KUKA KRL program: Work_2.src, Work_2.dat

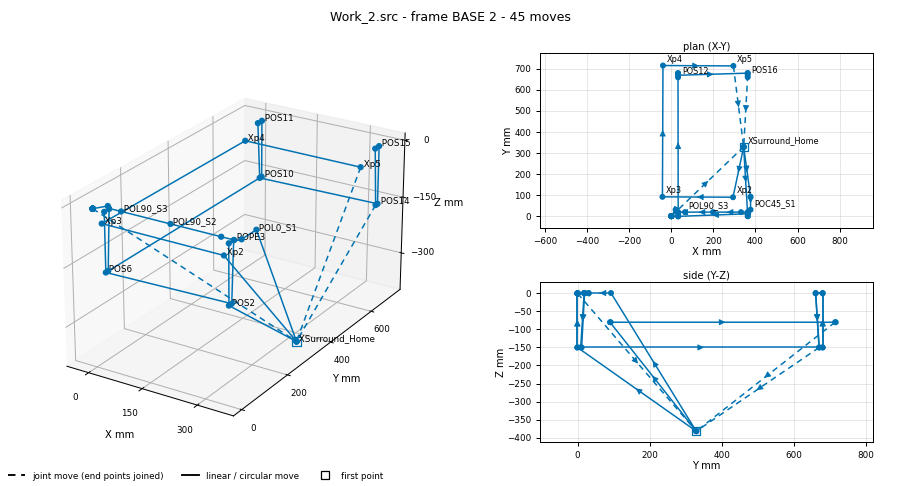
[picture p0: tool path of Work_2.src in frame BASE 2, 45 of 45 moves have a stored position in this frame; points joined in program order, loops and branches not executed]
--- Work_2.src ---
&ACCESS RVP
&REL 333
&PARAM EDITMASK = *
&PARAM TEMPLATE = C:\KRC\Roboter\Template\vorgabe
&PARAM DISKPATH = KRC:\R1\Program\HG
DEF Work_2( )
;FOLD INI;%{PE}
  ;FOLD BASISTECH INI
    GLOBAL INTERRUPT DECL 3 WHEN $STOPMESS==TRUE DO IR_STOPM ( )
    INTERRUPT ON 3
    BAS (#INITMOV,0 )
  ;ENDFOLD (BASISTECH INI)
  ;FOLD USER INI
    ;Make your modifications here

  ;ENDFOLD (USER INI)
;ENDFOLD (INI)

;FOLD Vision.Vision_Ini ;%{PE}%MKUKATPUSER




EKRL_Vision_Int_Data("Xml_Ini_Data")


;ENDFOLD
;loop
;FOLD PTP Surround_Home Vel=20 % PDAT1 Tool[2]:Work_Tool Base[2]:B_2;%{PE}%R 8.3.48,%MKUKATPBASIS,%CMOVE,%VPTP,%P 1:PTP, 2:Surround_Home, 3:, 5:20, 7:PDAT1
$BWDSTART=FALSE
PDAT_ACT=PPDAT1
FDAT_ACT=FSurround_Home
BAS(#PTP_PARAMS,20)
PTP XSurround_Home
;ENDFOLD

;FOLD Vision.Camera_Offset Camera_NAME :P2, Area:45, Work:2;%{PE}%MKUKATPUSER

 HanGao_Camera_Offset(#Calibration ,1,2,XP2)





;ENDFOLD
;FOLD LIN p2 Vel=.3 m/s CPDAT1 Tool[2]:Work_Tool Base[2]:B_2;%{PE}%R 8.3.48,%MKUKATPBASIS,%CMOVE,%VLIN,%P 1:LIN, 2:p2, 3:, 5:.3, 7:CPDAT1
$BWDSTART=FALSE
LDAT_ACT=LCPDAT1
FDAT_ACT=Fp2
BAS(#CP_PARAMS,.3)
LIN Xp2
;ENDFOLD
;FOLD Vision.Find_Model Work:2, Area:45;%{PE}%MKUKATPUSER



EKRL_Find_Model_Send("Xml_Vision_Model",2,1)



;ENDFOLD


;FOLD Vision.Camera_Offset Camera_NAME :P3, Area:135, Work:2;%{PE}%MKUKATPUSER

 HanGao_Camera_Offset(#Calibration ,2,2,XP3)





;ENDFOLD
;FOLD LIN p3 Vel=.3 m/s CPDAT2 Tool[2]:Work_Tool Base[2]:B_2;%{PE}%R 8.3.48,%MKUKATPBASIS,%CMOVE,%VLIN,%P 1:LIN, 2:p3, 3:, 5:.3, 7:CPDAT2
$BWDSTART=FALSE
LDAT_ACT=LCPDAT2
FDAT_ACT=Fp3
BAS(#CP_PARAMS,.3)
LIN Xp3
;ENDFOLD
;FOLD Vision.Find_Model Work:2, Area:135;%{PE}%MKUKATPUSER



EKRL_Find_Model_Send("Xml_Vision_Model",2,2)



;ENDFOLD


;FOLD Vision.Camera_Offset Camera_NAME :P4, Area:225, Work:2;%{PE}%MKUKATPUSER

 HanGao_Camera_Offset(#Calibration ,3,2,XP4)





;ENDFOLD
;FOLD LIN p4 Vel=.3 m/s CPDAT3 Tool[2]:Work_Tool Base[2]:B_2;%{PE}%R 8.3.48,%MKUKATPBASIS,%CMOVE,%VLIN,%P 1:LIN, 2:p4, 3:, 5:.3, 7:CPDAT3
$BWDSTART=FALSE
LDAT_ACT=LCPDAT3
FDAT_ACT=Fp4
BAS(#CP_PARAMS,.3)
LIN Xp4
;ENDFOLD
;FOLD Vision.Find_Model Work:2, Area:225;%{PE}%MKUKATPUSER



EKRL_Find_Model_Send("Xml_Vision_Model",2,3)



;ENDFOLD


;FOLD Vision.Camera_Offset Camera_NAME :P5, Area:315, Work:2;%{PE}%MKUKATPUSER

 HanGao_Camera_Offset(#Calibration ,4,2,XP5)





;ENDFOLD
;FOLD LIN p5 Vel=.3 m/s CPDAT4 Tool[2]:Work_Tool Base[2]:B_2;%{PE}%R 8.3.48,%MKUKATPBASIS,%CMOVE,%VLIN,%P 1:LIN, 2:p5, 3:, 5:.3, 7:CPDAT4
$BWDSTART=FALSE
LDAT_ACT=LCPDAT4
FDAT_ACT=Fp5
BAS(#CP_PARAMS,.3)
LIN Xp5
;ENDFOLD
;FOLD Vision.Find_Model Work:2, Area:315;%{PE}%MKUKATPUSER



EKRL_Find_Model_Send("Xml_Vision_Model",2,4)



;ENDFOLD
;endloop
;halt
;FOLD PTP Surround_Home Vel=10 % PDAT4 Tool[2]:Work_Tool Base[2]:B_2;%{PE}%R 8.3.48,%MKUKATPBASIS,%CMOVE,%VPTP,%P 1:PTP, 2:Surround_Home, 3:, 5:10, 7:PDAT4
$BWDSTART=FALSE
PDAT_ACT=PPDAT4
FDAT_ACT=FSurround_Home
BAS(#PTP_PARAMS,10)
PTP XSurround_Home
;ENDFOLD
;FOLD Surround_LIN.S_LIN Point:L0_S1, Vel=.2m/s, Point: 90/%, Area:LO, LDAT:L0_L1, OFFSET_NO:1, Work: N_2;%{PE}%MKUKATPUSER

; LIN L0_S1POS: X=0, Y=0, Z=0, A=0, B=0, C=0
; LIN Offset POS:X=0, Y=0, Z=0
HanGao_Surr_Calculate( 90, #L0, #L_LIN_POS , POL0_S1, , , L0_Welding_Craft[2,1].Welding_Offset  , , 1, 2 )

LL0_L1.VEL=L0_Welding_Craft[2,1].Welding_Speed
LL0_L1.ACC=L0_Welding_Craft[2,1].Welding_ACC
LL0_L1.APO_DIST=L0_Welding_Craft[2,1].Welding_CDIS

FDAT_ACT=FL0_S1
LDAT_ACT=LL0_L1
BAS(#CP_PARAMS,L0_Welding_Craft[2,1].Welding_Speed )
LIN POL0_S1 C_DIS C_DIS

;ENDFOLD
;FOLD Laser_Function.LSON POW= .9%, Sec= 0S;%{PE}%MKUKATPUSER


  $ANOUT[1]= .9
  LSON(0)


;ENDFOLD
;FOLD Surround_LIN.S_C_LIN Point:C45_S1, Vel=.04m/s, Area: C45, LDAT:C45_L1, Work: N_2;%{PE}%MKUKATPUSER

; CIR C45_S1POS: X=0, Y=0, Z=0, A=0, B=0, C=0
; CIR Offset POS:X=0, Y=0, Z=0
HanGao_Surr_Calculate(  , #C45, #C_LIN_POS , POC45_S1, , , C45_Welding_Craft[2,1].Welding_Offset , ,  , 2)

LC45_L1.VEL=C45_Welding_Craft[2,1].Welding_Speed
LC45_L1.ACC=C45_Welding_Craft[2,1].Welding_ACC
LC45_L1.APO_DIST=C45_Welding_Craft[2,1].Welding_CDIS

FDAT_ACT=FC45_S1
LDAT_ACT=LC45_L1
BAS(#CP_PARAMS, C45_Welding_Craft[2,1].Welding_Speed )
LIN POC45_S1 C_DIS C_DIS

;ENDFOLD
;FOLD Surround_CIR.S_C_CIR Point:PM3, PE3, Vel=.04m/s, Angle Area: C45, Work: N_2;%{PE}%MKUKATPUSER

; CIR MID POS:PM3 : X=0, Y=0, Z=0, A=0, B=0, C=0
; CIR END POS:PE3 : X=0, Y=0, Z=0, A=0, B=0, C=0
; CIR_MID_OFFSET  : X=0, Y=0, Z=0
; CIR_END_OFFSET  : X=0, Y=.3, Z=0
HanGao_Surr_Calculate(  , #C45, #C_CIR_POS ,  , POPM3, POPE3 , C45_Welding_Craft[2,2].Welding_Offset  , C45_Welding_Craft[2, 3].Welding_Offset  ,  , 2)

LPM3.VEL=C45_Welding_Craft[2,3].Welding_Speed
LPM3.ACC=C45_Welding_Craft[2,3].Welding_ACC
LPM3.APO_DIST=C45_Welding_Craft[2,3].Welding_CDIS

FDAT_ACT=FPE3
LDAT_ACT=LPM3
BAS(#CP_PARAMS,C45_Welding_Craft[2,3].Welding_Speed )
CIRC POPM3, POPE3 C_DIS C_DIS

;ENDFOLD
;FOLD Surround_LIN.S_LIN Point:L90_S1, Vel=.04m/s, Point: 10/%, Area:L90, LDAT:L90_L1, OFFSET_NO:1, Work: N_2;%{PE}%MKUKATPUSER

; LIN L90_S1POS: X=0, Y=0, Z=0, A=0, B=0, C=0
; LIN Offset POS:X=0, Y=.2, Z=0
HanGao_Surr_Calculate( 10, #L90, #L_LIN_POS , POL90_S1, , , L90_Welding_Craft[2,1].Welding_Offset  , , 1, 2 )

LL90_L1.VEL=L90_Welding_Craft[2,1].Welding_Speed
LL90_L1.ACC=L90_Welding_Craft[2,1].Welding_ACC
LL90_L1.APO_DIST=L90_Welding_Craft[2,1].Welding_CDIS

FDAT_ACT=FL90_S1
LDAT_ACT=LL90_L1
BAS(#CP_PARAMS,L90_Welding_Craft[2,1].Welding_Speed )
LIN POL90_S1 C_DIS C_DIS

;ENDFOLD
;FOLD Surround_LIN.S_LIN Point:L90_S2, Vel=.04m/s, Point: 50/%, Area:L90, LDAT:L90_L2, OFFSET_NO:2, Work: N_2;%{PE}%MKUKATPUSER

; LIN L90_S2POS: X=198.086502, Y=19.0685, Z=1, A=0, B=0, C=20
; LIN Offset POS:X=0, Y=.2, Z=0
HanGao_Surr_Calculate( 50, #L90, #L_LIN_POS , POL90_S2, , , L90_Welding_Craft[2,2].Welding_Offset  , , 2, 2 )

LL90_L2.VEL=L90_Welding_Craft[2,2].Welding_Speed
LL90_L2.ACC=L90_Welding_Craft[2,2].Welding_ACC
LL90_L2.APO_DIST=L90_Welding_Craft[2,2].Welding_CDIS

FDAT_ACT=FL90_S2
LDAT_ACT=LL90_L2
BAS(#CP_PARAMS,L90_Welding_Craft[2,2].Welding_Speed )
LIN POL90_S2 C_DIS C_DIS

;ENDFOLD
;FOLD Surround_LIN.S_LIN Point:L90_S3, Vel=.04m/s, Point: 90/%, Area:L90, LDAT:L90_L3, OFFSET_NO:3, Work: N_2;%{PE}%MKUKATPUSER

; LIN L90_S3POS: X=64.8645, Y=19.0867844, Z=1, A=0, B=0, C=20
; LIN Offset POS:X=0, Y=.2, Z=0
HanGao_Surr_Calculate( 90, #L90, #L_LIN_POS , POL90_S3, , , L90_Welding_Craft[2,3].Welding_Offset  , , 3, 2 )

LL90_L3.VEL=L90_Welding_Craft[2,3].Welding_Speed
LL90_L3.ACC=L90_Welding_Craft[2,3].Welding_ACC
LL90_L3.APO_DIST=L90_Welding_Craft[2,3].Welding_CDIS

FDAT_ACT=FL90_S3
LDAT_ACT=LL90_L3
BAS(#CP_PARAMS,L90_Welding_Craft[2,3].Welding_Speed )
LIN POL90_S3 C_DIS C_DIS

;ENDFOLD
;FOLD Surround_LIN.S_C_LIN Point:C135_S1, Vel=.04m/s, Area: C135, LDAT:C135_L1, Work: N_2;%{PE}%MKUKATPUSER

; CIR C135_S1POS: X=31.5589905, Y=18.8913536, Z=1, A=0, B=0, C=20
; CIR Offset POS:X=0, Y=.2, Z=0
HanGao_Surr_Calculate(  , #C135, #C_LIN_POS , POC135_S1, , , C135_Welding_Craft[2,1].Welding_Offset , ,  , 2)

LC135_L1.VEL=C135_Welding_Craft[2,1].Welding_Speed
LC135_L1.ACC=C135_Welding_Craft[2,1].Welding_ACC
LC135_L1.APO_DIST=C135_Welding_Craft[2,1].Welding_CDIS

FDAT_ACT=FC135_S1
LDAT_ACT=LC135_L1
BAS(#CP_PARAMS, C135_Welding_Craft[2,1].Welding_Speed )
LIN POC135_S1 C_DIS C_DIS

;ENDFOLD
;FOLD Surround_CIR.S_C_CIR Point:PM4, PE4, Vel=.04m/s, Angle Area: C135, Work: N_2;%{PE}%MKUKATPUSER

; CIR MID POS:PM4 : X=22.393, Y=22.49, Z=1, A=0, B=0, C=0
; CIR END POS:PE4 : X=20.0512314, Y=30.8929977, Z=0, A=0, B=-20, C=0
; CIR_MID_OFFSET  : X=0, Y=0, Z=0
; CIR_END_OFFSET  : X=.5, Y=0, Z=-1
HanGao_Surr_Calculate(  , #C135, #C_CIR_POS ,  , POPM4, POPE4 , C135_Welding_Craft[2,2].Welding_Offset  , C135_Welding_Craft[2, 3].Welding_Offset  ,  , 2)

LPM4.VEL=C135_Welding_Craft[2,3].Welding_Speed
LPM4.ACC=C135_Welding_Craft[2,3].Welding_ACC
LPM4.APO_DIST=C135_Welding_Craft[2,3].Welding_CDIS

FDAT_ACT=FPE4
LDAT_ACT=LPM4
BAS(#CP_PARAMS,C135_Welding_Craft[2,3].Welding_Speed )
CIRC POPM4, POPE4 C_DIS C_DIS

;ENDFOLD
;FOLD Surround_LIN.S_LIN Point:L180_S1, Vel=.04m/s, Point: 10/%, Area:L180, LDAT:L180_L1, OFFSET_NO:1, Work: N_2;%{PE}%MKUKATPUSER

; LIN L180_S1POS: X=19.5112858, Y=92.5949936, Z=0, A=0, B=-20, C=0
; LIN Offset POS:X=0, Y=0, Z=-1
HanGao_Surr_Calculate( 10, #L180, #L_LIN_POS , POL180_S1, , , L180_Welding_Craft[2,1].Welding_Offset  , , 1, 2 )

LL180_L1.VEL=L180_Welding_Craft[2,1].Welding_Speed
LL180_L1.ACC=L180_Welding_Craft[2,1].Welding_ACC
LL180_L1.APO_DIST=L180_Welding_Craft[2,1].Welding_CDIS

FDAT_ACT=FL180_S1
LDAT_ACT=LL180_L1
BAS(#CP_PARAMS,L180_Welding_Craft[2,1].Welding_Speed )
LIN POL180_S1 C_DIS C_DIS

;ENDFOLD
;FOLD Surround_LIN.S_LIN Point:L180_S2, Vel=.04m/s, Point: 50/%, Area:L180, LDAT:L180_L2, OFFSET_NO:2, Work: N_2;%{PE}%MKUKATPUSER

; LIN L180_S2POS: X=0, Y=0, Z=0, A=0, B=0, C=0
; LIN Offset POS:X=0, Y=0, Z=-1
HanGao_Surr_Calculate( 50, #L180, #L_LIN_POS , POL180_S2, , , L180_Welding_Craft[2,2].Welding_Offset  , , 2, 2 )

LL180_L2.VEL=L180_Welding_Craft[2,2].Welding_Speed
LL180_L2.ACC=L180_Welding_Craft[2,2].Welding_ACC
LL180_L2.APO_DIST=L180_Welding_Craft[2,2].Welding_CDIS

FDAT_ACT=FL180_S2
LDAT_ACT=LL180_L2
BAS(#CP_PARAMS,L180_Welding_Craft[2,2].Welding_Speed )
LIN POL180_S2 C_DIS C_DIS

;ENDFOLD
;FOLD Surround_LIN.S_LIN Point:L180_S3, Vel=.04m/s, Point: 95/%, Area:L180, LDAT:L180_L3, OFFSET_NO:3, Work: N_2;%{PE}%MKUKATPUSER

; LIN L180_S3POS: X=0, Y=0, Z=0, A=0, B=0, C=0
; LIN Offset POS:X=.5, Y=0, Z=-1
HanGao_Surr_Calculate( 95, #L180, #L_LIN_POS , POL180_S3, , , L180_Welding_Craft[2,3].Welding_Offset  , , 3, 2 )

LL180_L3.VEL=L180_Welding_Craft[2,3].Welding_Speed
LL180_L3.ACC=L180_Welding_Craft[2,3].Welding_ACC
LL180_L3.APO_DIST=L180_Welding_Craft[2,3].Welding_CDIS

FDAT_ACT=FL180_S3
LDAT_ACT=LL180_L3
BAS(#CP_PARAMS,L180_Welding_Craft[2,3].Welding_Speed )
LIN POL180_S3 C_DIS C_DIS

;ENDFOLD
;FOLD Surround_LIN.S_C_LIN Point:C225_S1, Vel=.04m/s, Area: C225, LDAT:C225_L1, Work: N_2;%{PE}%MKUKATPUSER

; CIR C225_S1POS: X=0, Y=0, Z=0, A=0, B=0, C=0
; CIR Offset POS:X=.5, Y=0, Z=-1
HanGao_Surr_Calculate(  , #C225, #C_LIN_POS , POC225_S1, , , C225_Welding_Craft[2,1].Welding_Offset , ,  , 2)

LC225_L1.VEL=C225_Welding_Craft[2,1].Welding_Speed
LC225_L1.ACC=C225_Welding_Craft[2,1].Welding_ACC
LC225_L1.APO_DIST=C225_Welding_Craft[2,1].Welding_CDIS

FDAT_ACT=FC225_S1
LDAT_ACT=LC225_L1
BAS(#CP_PARAMS, C225_Welding_Craft[2,1].Welding_Speed )
LIN POC225_S1 C_DIS C_DIS

;ENDFOLD
;FOLD Surround_CIR.S_C_CIR Point:PM5, PE5, Vel=.04m/s, Angle Area: C225, Work: N_2;%{PE}%MKUKATPUSER

; CIR MID POS:PM5 : X=22.393, Y=22.49, Z=1, A=0, B=0, C=0
; CIR END POS:PE5 : X=20.0512314, Y=30.8929977, Z=0, A=0, B=-20, C=0
; CIR_MID_OFFSET  : X=0, Y=0, Z=0
; CIR_END_OFFSET  : X=.5, Y=0, Z=-1
HanGao_Surr_Calculate(  , #C225, #C_CIR_POS ,  , POPM5, POPE5 , C225_Welding_Craft[2,2].Welding_Offset  , C225_Welding_Craft[2, 3].Welding_Offset  ,  , 2)

LPM5.VEL=C225_Welding_Craft[2,3].Welding_Speed
LPM5.ACC=C225_Welding_Craft[2,3].Welding_ACC
LPM5.APO_DIST=C225_Welding_Craft[2,3].Welding_CDIS

FDAT_ACT=FPE5
LDAT_ACT=LPM5
BAS(#CP_PARAMS,C225_Welding_Craft[2,3].Welding_Speed )
CIRC POPM5, POPE5 C_DIS C_DIS

;ENDFOLD
;FOLD Surround_LIN.S_LIN Point:L270_S1, Vel=.04m/s, Point: 10/%, Area:L270, LDAT:l270_L1, OFFSET_NO:1, Work: N_2;%{PE}%MKUKATPUSER

; LIN L270_S1POS: X=0, Y=0, Z=0, A=0, B=0, C=0
; LIN Offset POS:X=0, Y=0, Z=-1
HanGao_Surr_Calculate( 10, #L270, #L_LIN_POS , POL270_S1, , , L270_Welding_Craft[2,1].Welding_Offset  , , 1, 2 )

Ll270_L1.VEL=L270_Welding_Craft[2,1].Welding_Speed
Ll270_L1.ACC=L270_Welding_Craft[2,1].Welding_ACC
Ll270_L1.APO_DIST=L270_Welding_Craft[2,1].Welding_CDIS

FDAT_ACT=FL270_S1
LDAT_ACT=Ll270_L1
BAS(#CP_PARAMS,L270_Welding_Craft[2,1].Welding_Speed )
LIN POL270_S1 C_DIS C_DIS

;ENDFOLD
;FOLD Surround_LIN.S_LIN Point:L270_S2, Vel=.04m/s, Point: 50/%, Area:L270, LDAT:L270_L2, OFFSET_NO:2, Work: N_2;%{PE}%MKUKATPUSER

; LIN L270_S2POS: X=0, Y=0, Z=0, A=0, B=0, C=0
; LIN Offset POS:X=0, Y=0, Z=0
HanGao_Surr_Calculate( 50, #L270, #L_LIN_POS , POL270_S2, , , L270_Welding_Craft[2,2].Welding_Offset  , , 2, 2 )

LL270_L2.VEL=L270_Welding_Craft[2,2].Welding_Speed
LL270_L2.ACC=L270_Welding_Craft[2,2].Welding_ACC
LL270_L2.APO_DIST=L270_Welding_Craft[2,2].Welding_CDIS

FDAT_ACT=FL270_S2
LDAT_ACT=LL270_L2
BAS(#CP_PARAMS,L270_Welding_Craft[2,2].Welding_Speed )
LIN POL270_S2 C_DIS C_DIS

;ENDFOLD
;FOLD Surround_LIN.S_LIN Point:L270_S3, Vel=.04m/s, Point: 95/%, Area:L270, LDAT:L270_L3, OFFSET_NO:3, Work: N_2;%{PE}%MKUKATPUSER

; LIN L270_S3POS: X=0, Y=0, Z=0, A=0, B=0, C=0
; LIN Offset POS:X=0, Y=-.8, Z=0
HanGao_Surr_Calculate( 95, #L270, #L_LIN_POS , POL270_S3, , , L270_Welding_Craft[2,3].Welding_Offset  , , 3, 2 )

LL270_L3.VEL=L270_Welding_Craft[2,3].Welding_Speed
LL270_L3.ACC=L270_Welding_Craft[2,3].Welding_ACC
LL270_L3.APO_DIST=L270_Welding_Craft[2,3].Welding_CDIS

FDAT_ACT=FL270_S3
LDAT_ACT=LL270_L3
BAS(#CP_PARAMS,L270_Welding_Craft[2,3].Welding_Speed )
LIN POL270_S3 C_DIS C_DIS

;ENDFOLD
;FOLD Surround_LIN.S_C_LIN Point:C315_S1, Vel=.04m/s, Area: C315, LDAT:C315_L1, Work: N_2;%{PE}%MKUKATPUSER

; CIR C315_S1POS: X=0, Y=0, Z=0, A=0, B=0, C=0
; CIR Offset POS:X=0, Y=-.8, Z=0
HanGao_Surr_Calculate(  , #C315, #C_LIN_POS , POC315_S1, , , C315_Welding_Craft[2,1].Welding_Offset , ,  , 2)

LC315_L1.VEL=C315_Welding_Craft[2,1].Welding_Speed
LC315_L1.ACC=C315_Welding_Craft[2,1].Welding_ACC
LC315_L1.APO_DIST=C315_Welding_Craft[2,1].Welding_CDIS

FDAT_ACT=FC315_S1
LDAT_ACT=LC315_L1
BAS(#CP_PARAMS, C315_Welding_Craft[2,1].Welding_Speed )
LIN POC315_S1 C_DIS C_DIS

;ENDFOLD
;FOLD Surround_CIR.S_C_CIR Point:PM7, PE7, Vel=.04m/s, Angle Area: C315, Work: N_2;%{PE}%MKUKATPUSER

; CIR MID POS:PM7 : X=0, Y=0, Z=0, A=0, B=0, C=0
; CIR END POS:PE7 : X=0, Y=0, Z=0, A=0, B=0, C=0
; CIR_MID_OFFSET  : X=0, Y=0, Z=0
; CIR_END_OFFSET  : X=0, Y=.5, Z=0
HanGao_Surr_Calculate(  , #C315, #C_CIR_POS ,  , POPM7, POPE7 , C315_Welding_Craft[2,2].Welding_Offset  , C315_Welding_Craft[2, 3].Welding_Offset  ,  , 2)

LPM7.VEL=C315_Welding_Craft[2,3].Welding_Speed
LPM7.ACC=C315_Welding_Craft[2,3].Welding_ACC
LPM7.APO_DIST=C315_Welding_Craft[2,3].Welding_CDIS

FDAT_ACT=FPE7
LDAT_ACT=LPM7
BAS(#CP_PARAMS,C315_Welding_Craft[2,3].Welding_Speed )
CIRC POPM7, POPE7 C_DIS C_DIS

;ENDFOLD
;FOLD Surround_LIN.S_LIN Point:L0_S2, Vel=.04m/s, Point: 10/%, Area:LO, LDAT:L0_L2, OFFSET_NO:2, Work: N_2;%{PE}%MKUKATPUSER

; LIN L0_S2POS: X=0, Y=0, Z=0, A=0, B=0, C=0
; LIN Offset POS:X=0, Y=0, Z=0
HanGao_Surr_Calculate( 10, #L0, #L_LIN_POS , POL0_S2, , , L0_Welding_Craft[2,2].Welding_Offset  , , 2, 2 )

LL0_L2.VEL=L0_Welding_Craft[2,2].Welding_Speed
LL0_L2.ACC=L0_Welding_Craft[2,2].Welding_ACC
LL0_L2.APO_DIST=L0_Welding_Craft[2,2].Welding_CDIS

FDAT_ACT=FL0_S2
LDAT_ACT=LL0_L2
BAS(#CP_PARAMS,L0_Welding_Craft[2,2].Welding_Speed )
LIN POL0_S2 C_DIS C_DIS

;ENDFOLD
;FOLD Surround_LIN.S_LIN Point:L0_S3, Vel=.04m/s, Point: 50/%, Area:LO, LDAT:L0_L3, OFFSET_NO:3, Work: N_2;%{PE}%MKUKATPUSER

; LIN L0_S3POS: X=0, Y=0, Z=0, A=0, B=0, C=0
; LIN Offset POS:X=0, Y=0, Z=0
HanGao_Surr_Calculate( 50, #L0, #L_LIN_POS , POL0_S3, , , L0_Welding_Craft[2,3].Welding_Offset  , , 3, 2 )

LL0_L3.VEL=L0_Welding_Craft[2,3].Welding_Speed
LL0_L3.ACC=L0_Welding_Craft[2,3].Welding_ACC
LL0_L3.APO_DIST=L0_Welding_Craft[2,3].Welding_CDIS

FDAT_ACT=FL0_S3
LDAT_ACT=LL0_L3
BAS(#CP_PARAMS,L0_Welding_Craft[2,3].Welding_Speed )
LIN POL0_S3 C_DIS C_DIS

;ENDFOLD
;FOLD Surround_LIN.S_LIN Point:L0_S4, Vel=.04m/s, Point: 95/%, Area:LO, LDAT:L0_L4, OFFSET_NO:4, Work: N_2;%{PE}%MKUKATPUSER

; LIN L0_S4POS: X=0, Y=0, Z=0, A=0, B=0, C=0
; LIN Offset POS:X=0, Y=0, Z=0
HanGao_Surr_Calculate( 95, #L0, #L_LIN_POS , POL0_S4, , , L0_Welding_Craft[2,4].Welding_Offset  , , 4, 2 )

LL0_L4.VEL=L0_Welding_Craft[2,4].Welding_Speed
LL0_L4.ACC=L0_Welding_Craft[2,4].Welding_ACC
LL0_L4.APO_DIST=L0_Welding_Craft[2,4].Welding_CDIS

FDAT_ACT=FL0_S4
LDAT_ACT=LL0_L4
BAS(#CP_PARAMS,L0_Welding_Craft[2,4].Welding_Speed )
LIN POL0_S4 C_DIS C_DIS

;ENDFOLD
LSOFF()


;FOLD PTP Surround_Home Vel=10 % PDAT2 Tool[2]:Work_Tool Base[2]:B_2;%{PE}%R 8.3.48,%MKUKATPBASIS,%CMOVE,%VPTP,%P 1:PTP, 2:Surround_Home, 3:, 5:10, 7:PDAT2
$BWDSTART=FALSE
PDAT_ACT=PPDAT2
FDAT_ACT=FSurround_Home
BAS(#PTP_PARAMS,10)
PTP XSurround_Home
;ENDFOLD
if (false) THEN
;halt
;return
;FOLD Short_Craft.S_LIN Point:S2, Vel=.1m/s, Area: N45, Short_Pos: Safety, Point: 50/%, LDAT:L2, Work: N_2;%{PE}%MKUKATPUSER

; LIN S2POS: X=364.543579, Y=6.21706629, Z=0, A=0, B=0, C=0
; LIN Offset POS:X=0, Y=0, Z=0
HanGao_Surr_Calculate( 50, #N45, #L_LIN_POS , POS2, , , N45_Short_Craft[2,1].Welding_Offset  , , 1, 2, N2_Sink_Data.Sink_Type)

FDAT_ACT=FS2
LDAT_ACT=LL2
BAS(#CP_PARAMS,N45_Short_Craft[2,1].Welding_Speed )
LIN POS2 C_DIS C_DIS

;ENDFOLD
;FOLD Short_Craft.S_LIN Point:S3, Vel=.1m/s, Area: N45, Short_Pos: Start, Point: 50/%, LDAT:L3, Work: N_2;%{PE}%MKUKATPUSER

; LIN S3POS: X=0, Y=0, Z=0, A=0, B=0, C=0
; LIN Offset POS:X=0, Y=0, Z=0
HanGao_Surr_Calculate( 50, #N45, #L_LIN_POS , POS3, , , N45_Short_Craft[2,2].Welding_Offset  , , 2, 2, N2_Sink_Data.Sink_Type)

FDAT_ACT=FS3
LDAT_ACT=LL3
BAS(#CP_PARAMS,N45_Short_Craft[2,2].Welding_Speed )
LIN POS3 C_DIS C_DIS

;ENDFOLD
;FOLD ANOUT AO01=.6 ;%{PE}%R 8.3.48,%MKUKATPBASIS,%CANA,%VANOUT_STAT,%P 2:CHANNEL_1, 4:.6
$ANOUT[1]=.6
;ENDFOLD
LSON()
;FOLD Short_Craft.S_LIN Point:S4, Vel=.1m/s, Area: N45, Short_Pos: End, Point: 50/%, LDAT:L4, Work: N_2;%{PE}%MKUKATPUSER

; LIN S4POS: X=364.543579, Y=6.21706629, Z=0, A=0, B=0, C=0
; LIN Offset POS:X=0, Y=0, Z=0
HanGao_Surr_Calculate( 50, #N45, #L_LIN_POS , POS4, , , N45_Short_Craft[2,3].Welding_Offset  , , 3, 2, N2_Sink_Data.Sink_Type)

FDAT_ACT=FS4
LDAT_ACT=LL4
BAS(#CP_PARAMS,N45_Short_Craft[2,3].Welding_Speed )
LIN POS4 C_DIS C_DIS

;ENDFOLD
;FOLD Short_Craft.S_LIN Point:S5, Vel=.1m/s, Area: N45, Short_Pos: BackWelding, Point: 10/%, LDAT:L5, Work: N_2;%{PE}%MKUKATPUSER

; LIN S5POS: X=364.551483, Y=29.6448097, Z=0, A=0, B=0, C=0
; LIN Offset POS:X=0, Y=0, Z=0
HanGao_Surr_Calculate( 10, #N45, #L_LIN_POS , POS5, , , N45_Short_Craft[2,4].Welding_Offset  , , 4, 2, N2_Sink_Data.Sink_Type)

FDAT_ACT=FS5
LDAT_ACT=LL5
BAS(#CP_PARAMS,N45_Short_Craft[2,4].Welding_Speed )
LIN POS5 C_DIS C_DIS

;ENDFOLD
LSOFF()


;FOLD Short_Craft.S_LIN Point:S6, Vel=.1m/s, Area: N135, Short_Pos: Safety, Point: 50/%, LDAT:L6, Work: N_2;%{PE}%MKUKATPUSER

; LIN S6POS: X=364.547089, Y=16.5598412, Z=-150, A=0, B=0, C=0
; LIN Offset POS:X=0, Y=0, Z=0
HanGao_Surr_Calculate( 50, #N135, #L_LIN_POS , POS6, , , N135_Short_Craft[2,1].Welding_Offset  , , 1, 2, N2_Sink_Data.Sink_Type)

FDAT_ACT=FS6
LDAT_ACT=LL6
BAS(#CP_PARAMS,N135_Short_Craft[2,1].Welding_Speed )
LIN POS6 C_DIS C_DIS

;ENDFOLD
;FOLD Short_Craft.S_LIN Point:S7, Vel=.1m/s, Area: N135, Short_Pos: Start, Point: 50/%, LDAT:L7, Work: N_2;%{PE}%MKUKATPUSER

; LIN S7POS: X=36.6399193, Y=6.3348074, Z=-150, A=0, B=0, C=0
; LIN Offset POS:X=0, Y=0, Z=0
HanGao_Surr_Calculate( 50, #N135, #L_LIN_POS , POS7, , , N135_Short_Craft[2,2].Welding_Offset  , , 2, 2, N2_Sink_Data.Sink_Type)

FDAT_ACT=FS7
LDAT_ACT=LL7
BAS(#CP_PARAMS,N135_Short_Craft[2,2].Welding_Speed )
LIN POS7 C_DIS C_DIS

;ENDFOLD
;FOLD ANOUT AO01=.6 ;%{PE}%R 8.3.48,%MKUKATPBASIS,%CANA,%VANOUT_STAT,%P 2:CHANNEL_1, 4:.6
$ANOUT[1]=.6
;ENDFOLD
LSON()
;FOLD Short_Craft.S_LIN Point:S8, Vel=.1m/s, Area: N135, Short_Pos: End, Point: 50/%, LDAT:L8, Work: N_2;%{PE}%MKUKATPUSER

; LIN S8POS: X=36.6399193, Y=6.3348074, Z=0, A=0, B=0, C=0
; LIN Offset POS:X=0, Y=0, Z=0
HanGao_Surr_Calculate( 50, #N135, #L_LIN_POS , POS8, , , N135_Short_Craft[2,3].Welding_Offset  , , 3, 2, N2_Sink_Data.Sink_Type)

FDAT_ACT=FS8
LDAT_ACT=LL8
BAS(#CP_PARAMS,N135_Short_Craft[2,3].Welding_Speed )
LIN POS8 C_DIS C_DIS

;ENDFOLD
;FOLD Short_Craft.S_LIN Point:S9, Vel=.1m/s, Area: N135, Short_Pos: BackWelding, Point: 50/%, LDAT:L9, Work: N_2;%{PE}%MKUKATPUSER

; LIN S9POS: X=36.5802116, Y=29.963192, Z=0, A=0, B=0, C=0
; LIN Offset POS:X=0, Y=0, Z=0
HanGao_Surr_Calculate( 50, #N135, #L_LIN_POS , POS9, , , N135_Short_Craft[2,4].Welding_Offset  , , 4, 2, N2_Sink_Data.Sink_Type)

FDAT_ACT=FS9
LDAT_ACT=LL9
BAS(#CP_PARAMS,N135_Short_Craft[2,4].Welding_Speed )
LIN POS9 C_DIS C_DIS

;ENDFOLD
LSOFF()


;FOLD Short_Craft.S_LIN Point:S10, Vel=.1m/s, Area: N225, Short_Pos: Safety, Point: 50/%, LDAT:L10, Work: N_2;%{PE}%MKUKATPUSER

; LIN S10POS: X=36.6100655, Y=18.1489983, Z=-150, A=0, B=0, C=0
; LIN Offset POS:X=0, Y=0, Z=0
HanGao_Surr_Calculate( 50, #N225, #L_LIN_POS , POS10, , , N225_Short_Craft[2,1].Welding_Offset  , , 1, 2, N2_Sink_Data.Sink_Type)

FDAT_ACT=FS10
LDAT_ACT=LL10
BAS(#CP_PARAMS,N225_Short_Craft[2,1].Welding_Speed )
LIN POS10 C_DIS C_DIS

;ENDFOLD
;FOLD Short_Craft.S_LIN Point:S11, Vel=.1m/s, Area: N225, Short_Pos: Start, Point: 50/%, LDAT:L11, Work: N_2;%{PE}%MKUKATPUSER

; LIN S11POS: X=46.8049, Y=687.557678, Z=-150, A=0, B=0, C=0
; LIN Offset POS:X=0, Y=0, Z=0
HanGao_Surr_Calculate( 50, #N225, #L_LIN_POS , POS11, , , N225_Short_Craft[2,2].Welding_Offset  , , 2, 2, N2_Sink_Data.Sink_Type)

FDAT_ACT=FS11
LDAT_ACT=LL11
BAS(#CP_PARAMS,N225_Short_Craft[2,2].Welding_Speed )
LIN POS11 C_DIS C_DIS

;ENDFOLD
;FOLD ANOUT AO01=.6 ;%{PE}%R 8.3.48,%MKUKATPBASIS,%CANA,%VANOUT_STAT,%P 2:CHANNEL_1, 4:.6
$ANOUT[1]=.6
;ENDFOLD
LSON()
;FOLD Short_Craft.S_LIN Point:S12, Vel=.1m/s, Area: N225, Short_Pos: End, Point: 50/%, LDAT:L12, Work: N_2;%{PE}%MKUKATPUSER

; LIN S12POS: X=46.8049, Y=687.557678, Z=0, A=0, B=0, C=0
; LIN Offset POS:X=0, Y=0, Z=0
HanGao_Surr_Calculate( 50, #N225, #L_LIN_POS , POS12, , , N225_Short_Craft[2,3].Welding_Offset  , , 3, 2, N2_Sink_Data.Sink_Type)

FDAT_ACT=FS12
LDAT_ACT=LL12
BAS(#CP_PARAMS,N225_Short_Craft[2,3].Welding_Speed )
LIN POS12 C_DIS C_DIS

;ENDFOLD
;FOLD Short_Craft.S_LIN Point:S13, Vel=.1m/s, Area: N225, Short_Pos: BackWelding, Point: 50/%, LDAT:L13, Work: N_2;%{PE}%MKUKATPUSER

; LIN S13POS: X=46.2807388, Y=663.904114, Z=0, A=0, B=0, C=0
; LIN Offset POS:X=0, Y=0, Z=0
HanGao_Surr_Calculate( 50, #N225, #L_LIN_POS , POS13, , , N225_Short_Craft[2,4].Welding_Offset  , , 4, 2, N2_Sink_Data.Sink_Type)

FDAT_ACT=FS13
LDAT_ACT=LL13
BAS(#CP_PARAMS,N225_Short_Craft[2,4].Welding_Speed )
LIN POS13 C_DIS C_DIS

;ENDFOLD
LSOFF()


;FOLD Short_Craft.S_LIN Point:S14, Vel=.1m/s, Area: N315, Short_Pos: Safety, Point: 50/%, LDAT:L14, Work: N_2;%{PE}%MKUKATPUSER

; LIN S14POS: X=46.54282, Y=675.730896, Z=-150, A=0, B=0, C=0
; LIN Offset POS:X=0, Y=0, Z=0
HanGao_Surr_Calculate( 50, #N315, #L_LIN_POS , POS14, , , N315_Short_Craft[2,1].Welding_Offset  , , 1, 2, N2_Sink_Data.Sink_Type)

FDAT_ACT=FS14
LDAT_ACT=LL14
BAS(#CP_PARAMS,N315_Short_Craft[2,1].Welding_Speed )
LIN POS14 C_DIS C_DIS

;ENDFOLD
;FOLD Short_Craft.S_LIN Point:S15, Vel=.1m/s, Area: N315, Short_Pos: Start, Point: 50/%, LDAT:L15, Work: N_2;%{PE}%MKUKATPUSER

; LIN S15POS: X=375.074402, Y=680.748169, Z=-150, A=0, B=0, C=0
; LIN Offset POS:X=0, Y=0, Z=0
HanGao_Surr_Calculate( 50, #N315, #L_LIN_POS , POS15, , , N315_Short_Craft[2,2].Welding_Offset  , , 2, 2, N2_Sink_Data.Sink_Type)

FDAT_ACT=FS15
LDAT_ACT=LL15
BAS(#CP_PARAMS,N315_Short_Craft[2,2].Welding_Speed )
LIN POS15 C_DIS C_DIS

;ENDFOLD
;FOLD ANOUT AO01=.6 ;%{PE}%R 8.3.48,%MKUKATPBASIS,%CANA,%VANOUT_STAT,%P 2:CHANNEL_1, 4:.6
$ANOUT[1]=.6
;ENDFOLD
LSON()
;FOLD Short_Craft.S_LIN Point:S16, Vel=.1m/s, Area: N315, Short_Pos: End, Point: 50/%, LDAT:L16, Work: N_2;%{PE}%MKUKATPUSER

; LIN S16POS: X=375.074402, Y=680.748169, Z=0, A=0, B=0, C=0
; LIN Offset POS:X=0, Y=0, Z=0
HanGao_Surr_Calculate( 50, #N315, #L_LIN_POS , POS16, , , N315_Short_Craft[2,3].Welding_Offset  , , 3, 2, N2_Sink_Data.Sink_Type)

FDAT_ACT=FS16
LDAT_ACT=LL16
BAS(#CP_PARAMS,N315_Short_Craft[2,3].Welding_Speed )
LIN POS16 C_DIS C_DIS

;ENDFOLD
;FOLD Short_Craft.S_LIN Point:S17, Vel=.1m/s, Area: N315, Short_Pos: BackWelding, Point: 50/%, LDAT:L17, Work: N_2;%{PE}%MKUKATPUSER

; LIN S17POS: X=374.424377, Y=657.20105, Z=0, A=0, B=0, C=0
; LIN Offset POS:X=0, Y=0, Z=0
HanGao_Surr_Calculate( 50, #N315, #L_LIN_POS , POS17, , , N315_Short_Craft[2,4].Welding_Offset  , , 4, 2, N2_Sink_Data.Sink_Type)

FDAT_ACT=FS17
LDAT_ACT=LL17
BAS(#CP_PARAMS,N315_Short_Craft[2,4].Welding_Speed )
LIN POS17 C_DIS C_DIS

;ENDFOLD
LSOFF()
endif

;FOLD PTP Surround_Home CONT Vel=30 % PDAT3 Tool[2]:Work_Tool Base[2]:B_2;%{PE}%R 8.3.48,%MKUKATPBASIS,%CMOVE,%VPTP,%P 1:PTP, 2:Surround_Home, 3:C_DIS, 5:30, 7:PDAT3
$BWDSTART=FALSE
PDAT_ACT=PPDAT3
FDAT_ACT=FSurround_Home
BAS(#PTP_PARAMS,30)
PTP XSurround_Home C_DIS
;ENDFOLD
END

--- Work_2.dat ---
&ACCESS RVP
&REL 333
&PARAM EDITMASK = *
&PARAM TEMPLATE = C:\KRC\Roboter\Template\vorgabe
&PARAM DISKPATH = KRC:\R1\Program\HG
DEFDAT  Work_2
;FOLD EXTERNAL DECLARATIONS;%{PE}%MKUKATPBASIS,%CEXT,%VCOMMON,%P
;FOLD BASISTECH EXT;%{PE}%MKUKATPBASIS,%CEXT,%VEXT,%P
EXT  BAS (BAS_COMMAND  :IN,REAL  :IN )
DECL INT SUCCESS
;ENDFOLD (BASISTECH EXT)
;FOLD USER EXT;%{E}%MKUKATPUSER,%CEXT,%VEXT,%P
;Make your modifications here

;ENDFOLD (USER EXT)
;ENDFOLD (EXTERNAL DECLARATIONS)
DECL BASIS_SUGG_T LAST_BASIS={POINT1[] "P0                      ",POINT2[] "P0                      ",CP_PARAMS[] "CPDAT0                  ",PTP_PARAMS[] "PDAT0                   ",CONT[] "                        ",CP_VEL[] "2.0                     ",PTP_VEL[] " 100                    ",SYNC_PARAMS[] "SYNCDAT                 ",SPL_NAME[] "S0                      ",A_PARAMS[] "ADAT0                   "}
DECL E6POS XSURROUND_HOME={X 343.780548,Y 329.155823,Z -382.275,A 0.441927075,B -0.0416149125,C -0.0704164580,S 2,T 10,E1 0.0,E2 0.0,E3 0.0,E4 0.0,E5 0.0,E6 0.0}
DECL FDAT FSurround_Home={TOOL_NO 2,BASE_NO 2,IPO_FRAME #BASE,POINT2[] " ",TQ_STATE FALSE}
DECL PDAT PPDAT1={VEL 100.000,ACC 20.0000,APO_DIST 100.000,GEAR_JERK 50.0000,EXAX_IGN 0}
DECL PDAT PPDAT2={VEL 100.000,ACC 20.0000,APO_DIST 100.000,GEAR_JERK 50.0000,EXAX_IGN 0}
DECL E6POS POS2={X 363.220,Y -0.316000,Z -150.000,A 0.0,B 0.0,C 0.0}
DECL FDAT FS2={TOOL_NO 2,BASE_NO 2,IPO_FRAME #BASE,POINT2[] " ",TQ_STATE FALSE}
DECL LDAT LL2={VEL 0.100000,ACC 100.000,APO_DIST 5.00000,APO_FAC 50.0000,AXIS_VEL 100.000,AXIS_ACC 100.000,ORI_TYP #VAR,CIRC_TYP #BASE,JERK_FAC 50.0000,GEAR_JERK 50.0000,EXAX_IGN 0}
DECL E6POS POS3={X 363.220,Y -0.316000,Z 0.0,A 0.0,B 0.0,C 0.0}
DECL FDAT FS3={TOOL_NO 2,BASE_NO 2,IPO_FRAME #BASE,POINT2[] " ",TQ_STATE FALSE}
DECL LDAT LL3={VEL 0.100000,ACC 100.000,APO_DIST 0.0,APO_FAC 50.0000,AXIS_VEL 100.000,AXIS_ACC 100.000,ORI_TYP #VAR,CIRC_TYP #BASE,JERK_FAC 50.0000,GEAR_JERK 50.0000,EXAX_IGN 0}
DECL E6POS POS4={X 363.395,Y 19.3140,Z 0.0,A 0.0,B 0.0,C 0.0}
DECL FDAT FS4={TOOL_NO 2,BASE_NO 2,IPO_FRAME #BASE,POINT2[] " ",TQ_STATE FALSE}
DECL LDAT LL4={VEL 0.100000,ACC 100.000,APO_DIST 0.0,APO_FAC 50.0000,AXIS_VEL 100.000,AXIS_ACC 100.000,ORI_TYP #VAR,CIRC_TYP #BASE,JERK_FAC 50.0000,GEAR_JERK 50.0000,EXAX_IGN 0}
DECL E6POS POS5={X 363.323059,Y 11.2466183,Z -150.000,A 0.0,B 0.0,C 0.0}
DECL FDAT FS5={TOOL_NO 2,BASE_NO 2,IPO_FRAME #BASE,POINT2[] " ",TQ_STATE FALSE}
DECL LDAT LL5={VEL 0.100000,ACC 100.000,APO_DIST 0.0,APO_FAC 50.0000,AXIS_VEL 100.000,AXIS_ACC 100.000,ORI_TYP #VAR,CIRC_TYP #BASE,JERK_FAC 50.0000,GEAR_JERK 50.0000,EXAX_IGN 0}
DECL E6POS POPM3={X 373.063,Y 22.4860,Z 1.00000,A 0.0,B 0.0,C 0.0}
DECL E6POS POPE3={X 364.614,Y 19.1456451,Z 1.00000,A 0.0,B 0.0,C 20.0000}
DECL FDAT FPE3={TOOL_NO 2,BASE_NO 2,IPO_FRAME #BASE,POINT2[] " ",TQ_STATE FALSE}
DECL LDAT LPM3={VEL 0.01000000,ACC 100.000,APO_DIST 5.00000,APO_FAC 50.0000,AXIS_VEL 100.000,AXIS_ACC 100.000,ORI_TYP #VAR,CIRC_TYP #BASE,JERK_FAC 50.0000,GEAR_JERK 50.0000,EXAX_IGN 0}
DECL E6POS POS6={X 32.5260,Y -0.971000,Z -150.000,A 0.0,B 0.0,C 0.0}
DECL FDAT FS6={TOOL_NO 2,BASE_NO 2,IPO_FRAME #BASE,POINT2[] " ",TQ_STATE FALSE}
DECL LDAT LL6={VEL 0.100000,ACC 100.000,APO_DIST 0.0,APO_FAC 50.0000,AXIS_VEL 100.000,AXIS_ACC 100.000,ORI_TYP #VAR,CIRC_TYP #BASE,JERK_FAC 50.0000,GEAR_JERK 50.0000,EXAX_IGN 0}
DECL E6POS POS7={X 32.5260,Y -0.971000,Z 0.0,A 0.0,B 0.0,C 0.0}
DECL FDAT FS7={TOOL_NO 2,BASE_NO 2,IPO_FRAME #BASE,POINT2[] " ",TQ_STATE FALSE}
DECL LDAT LL7={VEL 0.100000,ACC 100.000,APO_DIST 0.0,APO_FAC 50.0000,AXIS_VEL 100.000,AXIS_ACC 100.000,ORI_TYP #VAR,CIRC_TYP #BASE,JERK_FAC 50.0000,GEAR_JERK 50.0000,EXAX_IGN 0}
DECL E6POS POS8={X 32.3940,Y 18.1940,Z 0.0,A 0.0,B 0.0,C 0.0}
DECL FDAT FS8={TOOL_NO 2,BASE_NO 2,IPO_FRAME #BASE,POINT2[] " ",TQ_STATE FALSE}
DECL LDAT LL8={VEL 0.100000,ACC 100.000,APO_DIST 0.0,APO_FAC 50.0000,AXIS_VEL 100.000,AXIS_ACC 100.000,ORI_TYP #VAR,CIRC_TYP #BASE,JERK_FAC 50.0000,GEAR_JERK 50.0000,EXAX_IGN 0}
DECL E6POS POS9={X 32.4600,Y 8.61150074,Z -150.000,A 0.0,B 0.0,C 0.0}
DECL FDAT FS9={TOOL_NO 2,BASE_NO 2,IPO_FRAME #BASE,POINT2[] " ",TQ_STATE FALSE}
DECL LDAT LL9={VEL 0.100000,ACC 100.000,APO_DIST 0.0,APO_FAC 50.0000,AXIS_VEL 100.000,AXIS_ACC 100.000,ORI_TYP #VAR,CIRC_TYP #BASE,JERK_FAC 50.0000,GEAR_JERK 50.0000,EXAX_IGN 0}
DECL E6POS POPM4={X 22.3930,Y 22.4900,Z 1.00000,A 0.0,B 0.0,C 0.0}
DECL E6POS POPE4={X 20.0512314,Y 30.8929977,Z 0.0,A 0.0,B -20.0000,C 0.0}
DECL FDAT FPE4={TOOL_NO 2,BASE_NO 2,IPO_FRAME #BASE,POINT2[] " ",TQ_STATE FALSE}
DECL LDAT LPM4={VEL 0.0120000,ACC 100.000,APO_DIST 5.00000,APO_FAC 50.0000,AXIS_VEL 100.000,AXIS_ACC 100.000,ORI_TYP #VAR,CIRC_TYP #BASE,JERK_FAC 50.0000,GEAR_JERK 50.0000,EXAX_IGN 0}
DECL E6POS POPM5={X 0.0,Y 0.0,Z 0.0,A 0.0,B 0.0,C 0.0}
DECL E6POS POPE5={X 0.0,Y 0.0,Z 0.0,A 0.0,B 0.0,C 0.0}
DECL FDAT FPE5={TOOL_NO 2,BASE_NO 2,IPO_FRAME #BASE,POINT2[] " ",TQ_STATE FALSE}
DECL LDAT LPM5={VEL 0.0400000,ACC 100.000,APO_DIST 5.00000,APO_FAC 50.0000,AXIS_VEL 100.000,AXIS_ACC 100.000,ORI_TYP #VAR,CIRC_TYP #BASE,JERK_FAC 50.0000,GEAR_JERK 50.0000,EXAX_IGN 0}
DECL E6POS POPM7={X 0.0,Y 0.0,Z 0.0,A 0.0,B 0.0,C 0.0}
DECL E6POS POPE7={X 0.0,Y 0.0,Z 0.0,A 0.0,B 0.0,C 0.0}
DECL FDAT FPE7={TOOL_NO 2,BASE_NO 2,IPO_FRAME #BASE,POINT2[] " ",TQ_STATE FALSE}
DECL LDAT LPM7={VEL 0.0400000,ACC 100.000,APO_DIST 5.00000,APO_FAC 50.0000,AXIS_VEL 100.000,AXIS_ACC 100.000,ORI_TYP #VAR,CIRC_TYP #BASE,JERK_FAC 50.0000,GEAR_JERK 50.0000,EXAX_IGN 0}
DECL E6POS POS10={X 31.6330,Y 679.439,Z -150.000,A 0.0,B 0.0,C 0.0}
DECL FDAT FS10={TOOL_NO 2,BASE_NO 2,IPO_FRAME #BASE,POINT2[] " ",TQ_STATE FALSE}
DECL LDAT LL10={VEL 0.100000,ACC 100.000,APO_DIST 0.0,APO_FAC 50.0000,AXIS_VEL 100.000,AXIS_ACC 100.000,ORI_TYP #VAR,CIRC_TYP #BASE,JERK_FAC 50.0000,GEAR_JERK 50.0000,EXAX_IGN 0}
DECL E6POS POS11={X 31.6330,Y 679.439,Z 0.0,A 0.0,B 0.0,C 0.0}
DECL FDAT FS11={TOOL_NO 2,BASE_NO 2,IPO_FRAME #BASE,POINT2[] " ",TQ_STATE FALSE}
DECL LDAT LL11={VEL 0.100000,ACC 100.000,APO_DIST 0.0,APO_FAC 50.0000,AXIS_VEL 100.000,AXIS_ACC 100.000,ORI_TYP #VAR,CIRC_TYP #BASE,JERK_FAC 50.0000,GEAR_JERK 50.0000,EXAX_IGN 0}
DECL E6POS POS12={X 31.8670,Y 660.025,Z 0.0,A 0.0,B 0.0,C 0.0}
DECL FDAT FS12={TOOL_NO 2,BASE_NO 2,IPO_FRAME #BASE,POINT2[] " ",TQ_STATE FALSE}
DECL LDAT LL12={VEL 0.100000,ACC 100.000,APO_DIST 0.0,APO_FAC 50.0000,AXIS_VEL 100.000,AXIS_ACC 100.000,ORI_TYP #VAR,CIRC_TYP #BASE,JERK_FAC 50.0000,GEAR_JERK 50.0000,EXAX_IGN 0}
DECL E6POS POS13={X 31.7500,Y 669.732056,Z -150.000,A 0.0,B 0.0,C 0.0}
DECL FDAT FS13={TOOL_NO 2,BASE_NO 2,IPO_FRAME #BASE,POINT2[] " ",TQ_STATE FALSE}
DECL LDAT LL13={VEL 0.100000,ACC 100.000,APO_DIST 0.0,APO_FAC 50.0000,AXIS_VEL 100.000,AXIS_ACC 100.000,ORI_TYP #VAR,CIRC_TYP #BASE,JERK_FAC 50.0000,GEAR_JERK 50.0000,EXAX_IGN 0}
DECL E6POS POS14={X 362.986,Y 679.910,Z -150.000,A 0.0,B 0.0,C 0.0}
DECL FDAT FS14={TOOL_NO 2,BASE_NO 2,IPO_FRAME #BASE,POINT2[] " ",TQ_STATE FALSE}
DECL LDAT LL14={VEL 0.100000,ACC 100.000,APO_DIST 0.0,APO_FAC 50.0000,AXIS_VEL 100.000,AXIS_ACC 100.000,ORI_TYP #VAR,CIRC_TYP #BASE,JERK_FAC 50.0000,GEAR_JERK 50.0000,EXAX_IGN 0}
DECL E6POS POS15={X 362.986,Y 679.910,Z 1.00000,A 0.0,B 0.0,C 0.0}
DECL FDAT FS15={TOOL_NO 2,BASE_NO 2,IPO_FRAME #BASE,POINT2[] " ",TQ_STATE FALSE}
DECL LDAT LL15={VEL 0.100000,ACC 100.000,APO_DIST 0.0,APO_FAC 50.0000,AXIS_VEL 100.000,AXIS_ACC 100.000,ORI_TYP #VAR,CIRC_TYP #BASE,JERK_FAC 50.0000,GEAR_JERK 50.0000,EXAX_IGN 0}
DECL E6POS POS16={X 363.044,Y 660.468,Z 1.00000,A 0.0,B 0.0,C 0.0}
DECL FDAT FS16={TOOL_NO 2,BASE_NO 2,IPO_FRAME #BASE,POINT2[] " ",TQ_STATE FALSE}
DECL LDAT LL16={VEL 0.100000,ACC 100.000,APO_DIST 0.0,APO_FAC 50.0000,AXIS_VEL 100.000,AXIS_ACC 100.000,ORI_TYP #VAR,CIRC_TYP #BASE,JERK_FAC 50.0000,GEAR_JERK 50.0000,EXAX_IGN 0}
DECL E6POS POS17={X 363.015,Y 670.188965,Z -150.000,A 0.0,B 0.0,C 0.0}
DECL FDAT FS17={TOOL_NO 2,BASE_NO 2,IPO_FRAME #BASE,POINT2[] " ",TQ_STATE FALSE}
DECL LDAT LL17={VEL 0.100000,ACC 100.000,APO_DIST 0.0,APO_FAC 50.0000,AXIS_VEL 100.000,AXIS_ACC 100.000,ORI_TYP #VAR,CIRC_TYP #BASE,JERK_FAC 50.0000,GEAR_JERK 50.0000,EXAX_IGN 0}
DECL PDAT PPDAT3={VEL 100.000,ACC 20.0000,APO_DIST 100.000,APO_MODE #CDIS,GEAR_JERK 50.0000,EXAX_IGN 0}
DECL FDAT FL0_S2={TOOL_NO 2,BASE_NO 2,IPO_FRAME #BASE,POINT2[] " ",TQ_STATE FALSE}
DECL E6POS POL0_S2={X 0.0,Y 0.0,Z 0.0,A 0.0,B 0.0,C 0.0}
DECL FDAT FL0={TOOL_NO 2,BASE_NO 11,IPO_FRAME #BASE,POINT2[] " ",TQ_STATE FALSE}
DECL E6POS POL0_s4={X 0.0,Y 0.0,Z 0.0,A 0.0,B 0.0,C 0.0}
DECL FDAT FL0_s4={TOOL_NO 2,BASE_NO 2,IPO_FRAME #BASE,POINT2[] " ",TQ_STATE FALSE}
DECL E6POS POC45_S5={X 404.000,Y 36.0000,Z -1.00000,A 0.0,B 20.0000,C 0.0}
DECL FDAT FC45_S5={TOOL_NO 2,BASE_NO 11,IPO_FRAME #BASE,POINT2[] " ",TQ_STATE FALSE}
DECL E6POS POL0_S1={X 376.526398,Y 92.6378174,Z 1.00000,A 0.0,B 20.0000,C 0.0}
DECL FDAT FL0_S1={TOOL_NO 2,BASE_NO 2,IPO_FRAME #BASE,POINT2[] " ",TQ_STATE FALSE}
DECL E6POS POC45_S1={X 376.599762,Y 30.8439941,Z 1.00000,A 0.0,B 20.0000,C 0.0}
DECL FDAT FC45_S1={TOOL_NO 2,BASE_NO 2,IPO_FRAME #BASE,POINT2[] " ",TQ_STATE FALSE}
DECL LDAT LL0_L1={VEL 0.200000,ACC 50.0000,APO_DIST 5.00000,APO_FAC 50.0000,AXIS_VEL 100.000,AXIS_ACC 100.000,ORI_TYP #VAR,CIRC_TYP #BASE,JERK_FAC 50.0000,GEAR_JERK 50.0000,EXAX_IGN 0}
DECL LDAT LC45_L1={VEL 0.0250000,ACC 100.000,APO_DIST 5.00000,APO_FAC 50.0000,AXIS_VEL 100.000,AXIS_ACC 100.000,ORI_TYP #VAR,CIRC_TYP #BASE,JERK_FAC 50.0000,GEAR_JERK 50.0000,EXAX_IGN 0}
DECL E6POS POL90_S1={X 331.308502,Y 19.0502167,Z 1.00000,A 0.0,B 0.0,C 20.0000}
DECL FDAT FL90_S1={TOOL_NO 2,BASE_NO 2,IPO_FRAME #BASE,POINT2[] " ",TQ_STATE FALSE}
DECL LDAT LL90_L1={VEL 0.0250000,ACC 100.000,APO_DIST 5.00000,APO_FAC 50.0000,AXIS_VEL 100.000,AXIS_ACC 100.000,ORI_TYP #VAR,CIRC_TYP #BASE,JERK_FAC 50.0000,GEAR_JERK 50.0000,EXAX_IGN 0}
DECL E6POS POL90_S2={X 198.086502,Y 19.0685,Z 1.00000,A 0.0,B 0.0,C 20.0000}
DECL FDAT FL90_S2={TOOL_NO 2,BASE_NO 2,IPO_FRAME #BASE,POINT2[] " ",TQ_STATE FALSE}
DECL LDAT LL90_L2={VEL 0.0250000,ACC 100.000,APO_DIST 5.00000,APO_FAC 50.0000,AXIS_VEL 100.000,AXIS_ACC 100.000,ORI_TYP #VAR,CIRC_TYP #BASE,JERK_FAC 50.0000,GEAR_JERK 50.0000,EXAX_IGN 0}
DECL E6POS POL90_S3={X 64.8645,Y 19.0867844,Z 1.00000,A 0.0,B 0.0,C 20.0000}
DECL FDAT FL90_S3={TOOL_NO 2,BASE_NO 2,IPO_FRAME #BASE,POINT2[] " ",TQ_STATE FALSE}
DECL LDAT LL90_L3={VEL 0.0250000,ACC 100.000,APO_DIST 5.00000,APO_FAC 50.0000,AXIS_VEL 100.000,AXIS_ACC 100.000,ORI_TYP #VAR,CIRC_TYP #BASE,JERK_FAC 50.0000,GEAR_JERK 50.0000,EXAX_IGN 0}
DECL E6POS POC135_S1={X 31.5589905,Y 18.8913536,Z 1.00000,A 0.0,B 0.0,C 20.0000}
DECL FDAT FC135_S1={TOOL_NO 2,BASE_NO 2,IPO_FRAME #BASE,POINT2[] " ",TQ_STATE FALSE}
DECL LDAT LC135_L1={VEL 0.0250000,ACC 100.000,APO_DIST 5.00000,APO_FAC 50.0000,AXIS_VEL 100.000,AXIS_ACC 100.000,ORI_TYP #VAR,CIRC_TYP #BASE,JERK_FAC 50.0000,GEAR_JERK 50.0000,EXAX_IGN 0}
DECL E6POS POL180_S1={X 0.0,Y 0.0,Z 0.0,A 0.0,B 0.0,C 0.0}
DECL FDAT FL180_S1={TOOL_NO 2,BASE_NO 2,IPO_FRAME #BASE,POINT2[] " ",TQ_STATE FALSE}
DECL LDAT LL180_L1={VEL 0.0400000,ACC 100.000,APO_DIST 0.0,APO_FAC 50.0000,AXIS_VEL 100.000,AXIS_ACC 100.000,ORI_TYP #VAR,CIRC_TYP #BASE,JERK_FAC 50.0000,GEAR_JERK 50.0000,EXAX_IGN 0}
DECL E6POS POL180_S2={X 0.0,Y 0.0,Z 0.0,A 0.0,B 0.0,C 0.0}
DECL FDAT FL180_S2={TOOL_NO 2,BASE_NO 2,IPO_FRAME #BASE,POINT2[] " ",TQ_STATE FALSE}
DECL LDAT LL180_L2={VEL 0.0400000,ACC 100.000,APO_DIST 0.0,APO_FAC 50.0000,AXIS_VEL 100.000,AXIS_ACC 100.000,ORI_TYP #VAR,CIRC_TYP #BASE,JERK_FAC 50.0000,GEAR_JERK 50.0000,EXAX_IGN 0}
DECL E6POS POL180_S3={X 0.0,Y 0.0,Z 0.0,A 0.0,B 0.0,C 0.0}
DECL FDAT FL180_S3={TOOL_NO 2,BASE_NO 2,IPO_FRAME #BASE,POINT2[] " ",TQ_STATE FALSE}
DECL LDAT LL180_L3={VEL 0.0400000,ACC 100.000,APO_DIST 0.0,APO_FAC 50.0000,AXIS_VEL 100.000,AXIS_ACC 100.000,ORI_TYP #VAR,CIRC_TYP #BASE,JERK_FAC 50.0000,GEAR_JERK 50.0000,EXAX_IGN 0}
DECL E6POS POC225_S1={X 0.0,Y 0.0,Z 0.0,A 0.0,B 0.0,C 0.0}
DECL FDAT FC225_S1={TOOL_NO 2,BASE_NO 2,IPO_FRAME #BASE,POINT2[] " ",TQ_STATE FALSE}
DECL LDAT LC225_L1={VEL 0.0400000,ACC 100.000,APO_DIST 0.0,APO_FAC 50.0000,AXIS_VEL 100.000,AXIS_ACC 100.000,ORI_TYP #VAR,CIRC_TYP #BASE,JERK_FAC 50.0000,GEAR_JERK 50.0000,EXAX_IGN 0}
DECL E6POS POL270_S1={X 0.0,Y 0.0,Z 0.0,A 0.0,B 0.0,C 0.0}
DECL FDAT FL270_S1={TOOL_NO 2,BASE_NO 2,IPO_FRAME #BASE,POINT2[] " ",TQ_STATE FALSE}
DECL LDAT Ll270_L1={VEL 0.0400000,ACC 100.000,APO_DIST 0.0,APO_FAC 50.0000,AXIS_VEL 100.000,AXIS_ACC 100.000,ORI_TYP #VAR,CIRC_TYP #BASE,JERK_FAC 50.0000,GEAR_JERK 50.0000,EXAX_IGN 0}
DECL E6POS POL270_S2={X 0.0,Y 0.0,Z 0.0,A 0.0,B 0.0,C 0.0}
DECL FDAT FL270_S2={TOOL_NO 2,BASE_NO 2,IPO_FRAME #BASE,POINT2[] " ",TQ_STATE FALSE}
DECL LDAT LL270_L2={VEL 0.0400000,ACC 100.000,APO_DIST 0.0,APO_FAC 50.0000,AXIS_VEL 100.000,AXIS_ACC 100.000,ORI_TYP #VAR,CIRC_TYP #BASE,JERK_FAC 50.0000,GEAR_JERK 50.0000,EXAX_IGN 0}
DECL E6POS POL270_S3={X 0.0,Y 0.0,Z 0.0,A 0.0,B 0.0,C 0.0}
DECL FDAT FL270_S3={TOOL_NO 2,BASE_NO 2,IPO_FRAME #BASE,POINT2[] " ",TQ_STATE FALSE}
DECL LDAT LL270_L3={VEL 0.0400000,ACC 100.000,APO_DIST 0.0,APO_FAC 50.0000,AXIS_VEL 100.000,AXIS_ACC 100.000,ORI_TYP #VAR,CIRC_TYP #BASE,JERK_FAC 50.0000,GEAR_JERK 50.0000,EXAX_IGN 0}
DECL E6POS POC315_S1={X 0.0,Y 0.0,Z 0.0,A 0.0,B 0.0,C 0.0}
DECL FDAT FC315_S1={TOOL_NO 2,BASE_NO 2,IPO_FRAME #BASE,POINT2[] " ",TQ_STATE FALSE}
DECL LDAT LC315_L1={VEL 0.0400000,ACC 100.000,APO_DIST 0.0,APO_FAC 50.0000,AXIS_VEL 100.000,AXIS_ACC 100.000,ORI_TYP #VAR,CIRC_TYP #BASE,JERK_FAC 50.0000,GEAR_JERK 50.0000,EXAX_IGN 0}
DECL LDAT LL0_L2={VEL 0.0400000,ACC 100.000,APO_DIST 0.0,APO_FAC 50.0000,AXIS_VEL 100.000,AXIS_ACC 100.000,ORI_TYP #VAR,CIRC_TYP #BASE,JERK_FAC 50.0000,GEAR_JERK 50.0000,EXAX_IGN 0}
DECL E6POS POL0_S3={X 0.0,Y 0.0,Z 0.0,A 0.0,B 0.0,C 0.0}
DECL FDAT FL0_S3={TOOL_NO 2,BASE_NO 2,IPO_FRAME #BASE,POINT2[] " ",TQ_STATE FALSE}
DECL LDAT LL0_L3={VEL 0.0400000,ACC 100.000,APO_DIST 0.0,APO_FAC 50.0000,AXIS_VEL 100.000,AXIS_ACC 100.000,ORI_TYP #VAR,CIRC_TYP #BASE,JERK_FAC 50.0000,GEAR_JERK 50.0000,EXAX_IGN 0}
DECL LDAT LL0_L4={VEL 0.0400000,ACC 100.000,APO_DIST 0.0,APO_FAC 50.0000,AXIS_VEL 100.000,AXIS_ACC 100.000,ORI_TYP #VAR,CIRC_TYP #BASE,JERK_FAC 50.0000,GEAR_JERK 50.0000,EXAX_IGN 0}
DECL E6POS XP2={X 293.122131,Y 89.9176636,Z -80.0293961,A 0.441927075,B -0.0416149199,C -0.0704164207,S 2,T 10,E1 0.0,E2 0.0,E3 0.0,E4 0.0,E5 0.0,E6 0.0}
DECL FDAT Fp2={TOOL_NO 2,BASE_NO 2,IPO_FRAME #BASE,POINT2[] " ",TQ_STATE FALSE}
DECL LDAT LCPDAT1={VEL 2.00000,ACC 100.000,APO_DIST 100.000,APO_FAC 50.0000,AXIS_VEL 100.000,AXIS_ACC 100.000,ORI_TYP #VAR,CIRC_TYP #BASE,JERK_FAC 50.0000,GEAR_JERK 50.0000,EXAX_IGN 0}
DECL E6POS XP3={X -42.3839874,Y 91.8151550,Z -80.0254822,A 0.441927075,B -0.0416149236,C -0.0704165,S 2,T 10,E1 0.0,E2 0.0,E3 0.0,E4 0.0,E5 0.0,E6 0.0}
DECL FDAT Fp3={TOOL_NO 2,BASE_NO 2,IPO_FRAME #BASE,POINT2[] " ",TQ_STATE FALSE}
DECL LDAT LCPDAT2={VEL 2.00000,ACC 100.000,APO_DIST 100.000,APO_FAC 50.0000,AXIS_VEL 100.000,AXIS_ACC 100.000,ORI_TYP #VAR,CIRC_TYP #BASE,JERK_FAC 50.0000,GEAR_JERK 50.0000,EXAX_IGN 0}
DECL E6POS XP4={X -39.7999954,Y 716.082336,Z -80.0293350,A 0.441927075,B -0.0416149311,C -0.0704164803,S 2,T 10,E1 0.0,E2 0.0,E3 0.0,E4 0.0,E5 0.0,E6 0.0}
DECL FDAT Fp4={TOOL_NO 2,BASE_NO 2,IPO_FRAME #BASE,POINT2[] " ",TQ_STATE FALSE}
DECL LDAT LCPDAT3={VEL 2.00000,ACC 100.000,APO_DIST 100.000,APO_FAC 50.0000,AXIS_VEL 100.000,AXIS_ACC 100.000,ORI_TYP #VAR,CIRC_TYP #BASE,JERK_FAC 50.0000,GEAR_JERK 50.0000,EXAX_IGN 0}
DECL E6POS XP5={X 294.984924,Y 714.198059,Z -80.0293350,A 0.441927075,B -0.0416149311,C -0.0704164803,S 2,T 10,E1 0.0,E2 0.0,E3 0.0,E4 0.0,E5 0.0,E6 0.0}
DECL FDAT Fp5={TOOL_NO 2,BASE_NO 2,IPO_FRAME #BASE,POINT2[] " ",TQ_STATE FALSE}
DECL LDAT LCPDAT4={VEL 2.00000,ACC 100.000,APO_DIST 100.000,APO_FAC 50.0000,AXIS_VEL 100.000,AXIS_ACC 100.000,ORI_TYP #VAR,CIRC_TYP #BASE,JERK_FAC 50.0000,GEAR_JERK 50.0000,EXAX_IGN 0}
DECL PDAT PPDAT4={VEL 100.000,ACC 20.0000,APO_DIST 100.000,GEAR_JERK 50.0000,EXAX_IGN 0}
ENDDAT
